FUNCTION_BLOCK FB_SQRT (* Square root of a REAL value *)
  (* Standard: IEC 61499-1-D.1; Classification: Math functions; Function: Square root; Type: REAL *)
  (* Version 0.0, 2006-05-01, JHC, Holobloc Inc *)
  (* Compiler header: package fb.rt.math; *)
  (* Compiler classdef: class FB_SQRT extends FBFunction1 *)
  (* Compiler Java Sun JDK 1.5.0 *)
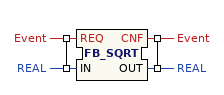
  EVENT_INPUT
    REQ WITH IN;
  END_EVENT
  EVENT_OUTPUT
    CNF WITH OUT;
  END_EVENT
  VAR_INPUT
    IN : REAL;
  END_VAR
  VAR_OUTPUT
    OUT : REAL; (* Converted value *)
  END_VAR
END_FUNCTION_BLOCK
